# EPICS autosave request: IOCs/12id/iocBoot/ioc12idb/auto_positions.req
$(P)m1.DVAL
$(P)m2.DVAL
$(P)m3.DVAL
$(P)m4.DVAL
$(P)m5.DVAL
$(P)m6.DVAL
$(P)m7.DVAL
$(P)m8.DVAL
$(P)m9.DVAL
$(P)m10.DVAL
$(P)m11.DVAL
$(P)m12.DVAL
$(P)m13.DVAL
$(P)m14.DVAL
$(P)m15.DVAL
$(P)m16.DVAL
$(P)m17.DVAL
$(P)m18.DVAL
$(P)m19.DVAL
$(P)m20.DVAL
$(P)m21.DVAL
$(P)m22.DVAL
$(P)m23.DVAL
$(P)m24.DVAL

$(P)SM1.DVAL
$(P)SM2.DVAL
$(P)SM3.DVAL
$(P)SM4.DVAL
$(P)SM5.DVAL
$(P)SM6.DVAL
$(P)SM7.DVAL
$(P)SM8.DVAL
$(P)SM9.DVAL
$(P)SM10.DVAL
